Staubli VAL3: encTrajPtAck.pgx

public program encTrajPtAck()
begin
  // Copyright (c) 2016, Ocado Technology - Robotics Research Team
  //
  // Licensed under the Apache License, Version 2.0 (the "License");
  // you may not use this file except in compliance with the License.
  // You may obtain a copy of the License at
  //
  //     http://www.apache.org/licenses/LICENSE-2.0
  //
  // Unless required by applicable law or agreed to in writing, software
  // distributed under the License is distributed on an "AS IS" BASIS,
  // WITHOUT WARRANTIES OR CONDITIONS OF ANY KIND, either express or implied.
  // See the License for the specific language governing permissions and
  // limitations under the License.
  // encode 'prefix' and 'header'
  // encode 'prefix' and 'header'
  call encPrefixHeader(rosTrajPtAck.prefix, rosTrajPtAck.header)
  // encode 'sequence' variable of body message (data)
  // logMsg("msg body: "+toString("", rosTrajPtAck.jointTrajPt.nSeq))
  toBinary(rosTrajPtAck.jointTrajPt.nSeq,1,"-4l",rosTrajPtAck.body.nData)
  // encodings of 'joints[10]', 'velocity' and 'duration' ignored to save CPU time, since values are all zeros
end
